// TIA Portal V19 export
TYPE "FeedMachine_Wng"
// stored: Access Published
   STRUCT
      NotAutReady { ExternalVisible := 'False'; ExternalWritable := 'False'} : Bool;
      MissingCnd_Bkw { ExternalVisible := 'False'; ExternalWritable := 'False'} : Bool;
      MissingCnd_Fwd { ExternalVisible := 'False'; ExternalWritable := 'False'} : Bool;
      Ax : "TAx_Warnings";
   END_STRUCT;
END_TYPE
